INTERFACE I_NodeWithProtection EXTENDS I_Node

METHOD PUBLIC PreExecuteCheck : HRESULT
VAR
END_VAR
END_METHOD

END_INTERFACE

(* stored: Version 1.1.0.1, ProductVersion 3.1.4024.12
   Itf I_NodeWithProtection: Id {fc27a325-17b7-0c6b-0331-163f27b63604}
   Method PreExecuteCheck: Id {b6462e5e-90fa-0567-2763-f34d2cdf0d62} *)
